Staubli VAL3: strFill.pgx

public program strFill(string x_sMessageIn, num x_nLenMessOut, string& x_sMessageOut[])
  local string l_sEmpty
  local num l_nLen
begin
  //-----------------------------------------------------------------------
  //Header begin
  //Description of program
  //  To add spaces if the length of x_sMessageIn is less than the
  //  x_nLenMessOut.If the length of x_sMessageIn is greater than
  //  x_nLenMessOut it will be truncated.
  //  如果x_sMessageIn的消息长度是少于x_nLenMessOut的，增加空格。
  //  如果x_sMessageIn的消息长度是大于x_nLenMessOut的，将会被截断。
  //Input parameters
  //  string x_sMessageIn :
  //    role : Message that you want to display
  //    作用：你想去显示的消息
  //  num x_nLenMessOut :
  //    role : Length of the message out
  //    作用：输出消息的长度
  //Output parameters
  //  string x_sMessageOut :
  //    role : Message with spaces after or truncated if the length
  //          x_sMessageIn is greater than x_nLenMessOut
  //    作用：如果长度x_sMessageIn大于x_nLenMessOut，消息使用空格或被截断
  //Example
  //  call strFill("hello",20,l_sMessOut)
  //
  //History
  //  Creation : 28-04-08 - f.Rob
  //Header end
  //-----------------------------------------------------------------------
  //Look for asian message
  if getDisplayLen(x_sMessageIn)<x_nLenMessOut
    //Insert some spaces 插入一些空格
    l_sEmpty="                                        "
    x_sMessageOut=x_sMessageIn
    //Length of the spaces to add  增加空格的长度
    l_nLen=(x_nLenMessOut-getDisplayLen(x_sMessageIn))
    call midPos(l_sEmpty,l_nLen,0,x_sMessageIn)
    x_sMessageOut=x_sMessageOut+x_sMessageIn
  else
    if getDisplayLen(x_sMessageIn)>x_nLenMessOut
      //Divide the string  分割字符串
      call midPos(x_sMessageIn,x_nLenMessOut,0,x_sMessageOut)
    else
      //They are the same
      x_sMessageOut=x_sMessageIn
    endIf
  endIf
end
